Staubli VAL3: insertDialog.pgx

public program insertDialog(string x_sMsg, num& x_nItem[], num x_nMin, num x_nMax)
  local num l_nStartLine
  local num l_nLine
  local num i
  local num l_nPX
  local num l_nPY
  local string l_sItem
  local string l_sMessage
  local string l_sEmpty
begin
  //
  // modify the x_sItem, using a min max range
  //
  if watch(bShowDialog==false,3)==false
    bShowDialog=false
    return
  else
    setMutex(bShowDialog)
    // clear the line
    call clear(0,13)
    // look for the comma
    if round(x_nItem)!=x_nItem
      l_sItem=toString(".2",x_nItem)
    else
      l_sItem=toString("",x_nItem)
    endIf
    // print the line
    l_sItem=x_sMsg+">"+l_sItem
    call stringCopy(l_sItem,sMessage)
    // divide the sentence
    call divideString(sMessage,l_nLine)
    l_nStartLine=round(5-l_nLine/2)
    // Start LINE
    call type(0,l_nStartLine-2,"┌──────────────────────────────────────┐")
    call type(0,l_nStartLine-1,"│                                      │")
    // write the message
    for i=0 to l_nLine
      //call type(,"                                      ")
      l_sMessage=sMessage[i]
      call typeCenter(i+l_nStartLine,l_sMessage,38,false)
      call type(0,l_nStartLine+i,"│"+l_sMessage+"│")
    endFor
    // end LINE
    call type(0,l_nStartLine+l_nLine+1,"│                                      │")
    call type(0,l_nStartLine+l_nLine+2,"└──────────────────────────────────────┘")
    l_nPX=find(l_sMessage,">")+2
    l_nPY=l_nStartLine+l_nLine
    // change the value
    call changeValue(x_nItem,x_nMin,x_nMax,l_nPX,l_nPY,l_sEmpty)
    //
    bShowDialog=false
    bUseRefresh=true
    //
  endIf
end
